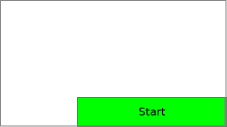
VISUALIZATION VIS_Main  // 227x127
    Button (77,97 150x30), "Start"
        tap SCADA_START
END_VISUALIZATION

(* stored: Version 1.1.0.1, ProductVersion 3.1.4026.18
   Visu VIS_Main: Id {594db05b-3253-49e6-81b3-d0df5bf2f443} *)
